Yaskawa INFORM job: malben_before.JBI

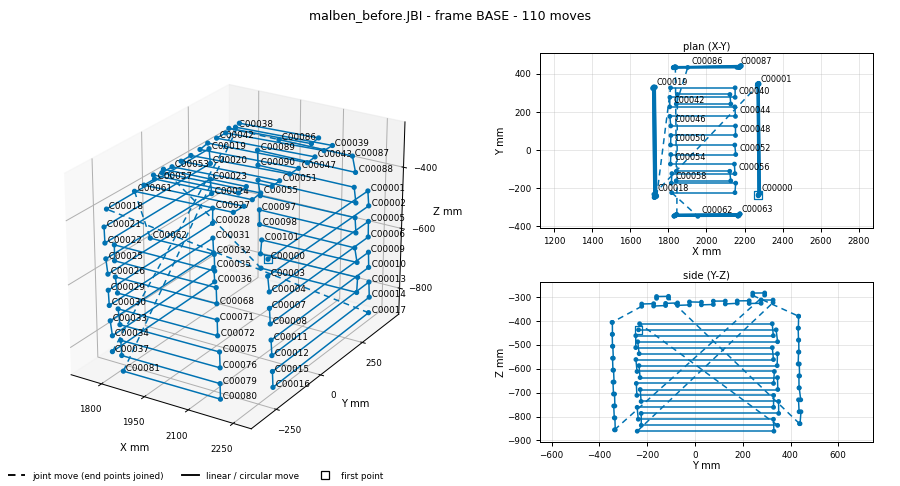
[picture p0: tool path of malben_before.JBI in frame BASE, 110 of 110 moves have a stored position in this frame; points joined in program order, loops and branches not executed]
/JOB
//NAME malben_before
//POS
///NPOS 110,0,0,0,0,0
///TOOL 0
///POSTYPE BASE
///RECTAN
///RCONF 1,0,0,0,0,0,0,0,0,0,0,0,0,0,0,0,0,0,0,0,0,0,0,0
C00000=2270.974700,-236.314400,-436.599200,0.000000,0.000000,0.000000
C00001=2266.659400,339.742100,-436.599200,0.000000,0.000000,0.000000
C00002=2267.434100,345.923800,-486.599200,0.000000,0.000000,0.000000
C00003=2272.441700,-239.676100,-486.599200,0.000000,0.000000,0.000000
C00004=2274.161000,-233.772700,-536.599200,0.000000,0.000000,0.000000
C00005=2268.116700,345.207300,-536.599200,0.000000,0.000000,0.000000
C00006=2269.414500,344.079000,-586.599200,0.000000,0.000000,0.000000
C00007=2275.422000,-234.403400,-586.599200,0.000000,0.000000,0.000000
C00008=2275.677100,-229.849900,-636.599200,0.000000,0.000000,0.000000
C00009=2270.908900,345.469500,-636.599200,0.000000,0.000000,0.000000
C00010=2272.247500,346.658600,-686.599200,0.000000,0.000000,0.000000
C00011=2278.345000,-229.368800,-686.599200,0.000000,0.000000,0.000000
C00012=2279.048100,-225.521500,-736.599200,0.000000,0.000000,0.000000
C00013=2272.572100,350.100400,-736.599200,0.000000,0.000000,0.000000
C00014=2274.809400,350.446800,-786.599200,0.000000,0.000000,0.000000
C00015=2281.061100,-225.219100,-786.599200,0.000000,0.000000,0.000000
C00016=2282.853200,-224.776000,-836.599200,0.000000,0.000000,0.000000
C00017=2276.307800,346.007400,-836.599200,0.000000,0.000000,0.000000
C00018=1724.578400,-231.807500,-411.083700,0.000000,90.000000,0.000000
C00019=1718.279300,323.447600,-411.083700,0.000000,90.000000,0.000000
C00020=1719.725400,327.955100,-461.083700,0.000000,90.000000,0.000000
C00021=1725.796900,-247.885600,-461.083700,0.000000,90.000000,0.000000
C00022=1727.476900,-248.031700,-511.083700,0.000000,90.000000,0.000000
C00023=1721.770500,323.709400,-511.083700,0.000000,90.000000,0.000000
C00024=1723.614500,328.610900,-561.083700,0.000000,90.000000,0.000000
C00025=1728.674900,-247.324100,-561.083700,0.000000,90.000000,0.000000
C00026=1731.265400,-242.598600,-611.083700,0.000000,90.000000,0.000000
C00027=1724.878400,332.404800,-611.083700,0.000000,90.000000,0.000000
C00028=1725.967100,328.907000,-661.083700,0.000000,90.000000,0.000000
C00029=1733.123300,-245.670000,-661.083700,0.000000,90.000000,0.000000
C00030=1733.584900,-243.188200,-711.083700,0.000000,90.000000,0.000000
C00031=1726.804300,329.270600,-711.083700,0.000000,90.000000,0.000000
C00032=1729.229800,328.994100,-761.083700,0.000000,90.000000,0.000000
C00033=1734.902000,-242.222300,-761.083700,0.000000,90.000000,0.000000
C00034=1737.913800,-237.463900,-811.083700,0.000000,90.000000,0.000000
C00035=1730.236300,328.580500,-811.083700,0.000000,90.000000,0.000000
C00036=1731.867100,330.516900,-861.083700,0.000000,90.000000,0.000000
C00037=1739.462300,-241.828500,-861.083700,0.000000,90.000000,0.000000
C00038=1812.070000,326.956500,-322.467000,-180.000000,0.000000,90.000000
C00039=2150.695600,326.956500,-312.028700,-180.000000,0.000000,90.000000
C00040=2150.727600,276.956500,-311.505300,-180.000000,0.000000,90.000000
C00041=1808.470300,276.956500,-325.644000,-180.000000,0.000000,90.000000
C00042=1807.754500,226.956500,-326.266200,-180.000000,0.000000,90.000000
C00043=2149.229600,226.956500,-314.851000,-180.000000,0.000000,90.000000
C00044=2152.427900,176.956500,-315.522800,-180.000000,0.000000,90.000000
C00045=1808.354700,176.956500,-325.499800,-180.000000,0.000000,90.000000
C00046=1813.127700,126.956500,-328.391500,-180.000000,0.000000,90.000000
C00047=2152.547100,126.956500,-316.102600,-180.000000,0.000000,90.000000
C00048=2152.688400,76.956500,-316.428000,-180.000000,0.000000,90.000000
C00049=1813.792200,76.956500,-330.537400,-180.000000,0.000000,90.000000
C00050=1812.079500,26.956500,-332.110200,-180.000000,0.000000,90.000000
C00051=2148.963600,26.956500,-320.940800,-180.000000,0.000000,90.000000
C00052=2153.965100,-23.043500,-319.751400,-180.000000,0.000000,90.000000
C00053=1813.274400,-23.043500,-332.397900,-180.000000,0.000000,90.000000
C00054=1811.443300,-73.043500,-334.201000,-180.000000,0.000000,90.000000
C00055=2146.917700,-73.043500,-323.945200,-180.000000,0.000000,90.000000
C00056=2149.738000,-123.043500,-326.004000,-180.000000,0.000000,90.000000
C00057=1819.062400,-123.043500,-334.939200,-180.000000,0.000000,90.000000
C00058=1816.212900,-173.043500,-337.150600,-180.000000,0.000000,90.000000
C00059=2153.683800,-173.043500,-327.184800,-180.000000,0.000000,90.000000
C00060=2149.816500,-223.043500,-328.439400,-180.000000,0.000000,90.000000
C00061=1817.967700,-223.043500,-338.250300,-180.000000,0.000000,90.000000
C00062=1954.986900,-347.317400,-405.440900,-90.000000,0.000000,0.000000
C00063=2165.301400,-346.003700,-405.440900,-90.000000,0.000000,0.000000
C00064=2166.306400,-345.533400,-455.440900,-90.000000,0.000000,0.000000
C00065=1831.008500,-346.423600,-455.440900,-90.000000,0.000000,0.000000
C00066=1829.824700,-345.452500,-505.440900,-90.000000,0.000000,0.000000
C00067=2169.877900,-343.987400,-505.440900,-90.000000,0.000000,0.000000
C00068=2170.261000,-341.942900,-555.440900,-90.000000,0.000000,0.000000
C00069=1830.845900,-345.180900,-555.440900,-90.000000,0.000000,0.000000
C00070=1835.840700,-343.537100,-605.440900,-90.000000,0.000000,0.000000
C00071=2170.679700,-340.902100,-605.440900,-90.000000,0.000000,0.000000
C00072=2170.579800,-338.805400,-655.440900,-90.000000,0.000000,0.000000
C00073=1836.308000,-343.283400,-655.440900,-90.000000,0.000000,0.000000
C00074=1839.916600,-341.222400,-705.440900,-90.000000,0.000000,0.000000
C00075=2175.279700,-336.688900,-705.440900,-90.000000,0.000000,0.000000
C00076=2176.238200,-335.487800,-755.440900,-90.000000,0.000000,0.000000
C00077=1840.835800,-340.227800,-755.440900,-90.000000,0.000000,0.000000
C00078=1841.292900,-337.885200,-805.440900,-90.000000,0.000000,0.000000
C00079=2175.716600,-335.286800,-805.440900,-90.000000,0.000000,0.000000
C00080=2175.900100,-333.842700,-855.440900,-90.000000,0.000000,0.000000
C00081=1845.052500,-336.997600,-855.440900,-90.000000,0.000000,0.000000
C00082=1847.834300,291.860000,-291.167300,-180.000000,0.000000,90.000000
C00083=2123.193800,291.860000,-282.202500,-180.000000,0.000000,90.000000
C00084=2127.968600,241.860000,-282.721100,-180.000000,0.000000,90.000000
C00085=1842.147700,241.860000,-292.609500,-180.000000,0.000000,90.000000
C00086=1902.222600,433.807700,-379.657800,90.000000,0.000000,0.000000
C00087=2160.048600,433.981200,-379.657800,90.000000,0.000000,0.000000
C00088=2172.433200,432.884400,-429.657800,90.000000,0.000000,0.000000
C00089=1826.230300,432.054000,-429.657800,90.000000,0.000000,0.000000
C00090=1827.301000,433.425300,-479.657800,90.000000,0.000000,0.000000
C00091=2168.117900,434.398200,-479.657800,90.000000,0.000000,0.000000
C00092=2174.981500,435.019500,-529.657800,90.000000,0.000000,0.000000
C00093=1827.672000,433.648700,-529.657800,90.000000,0.000000,0.000000
C00094=1837.169100,432.018700,-579.657800,90.000000,0.000000,0.000000
C00095=2172.360400,436.705800,-579.657800,90.000000,0.000000,0.000000
C00096=2175.918000,437.858200,-629.657800,90.000000,0.000000,0.000000
C00097=1832.142800,435.174100,-629.657800,90.000000,0.000000,0.000000
C00098=1832.804900,435.627000,-679.657800,90.000000,0.000000,0.000000
C00099=2173.854800,436.487800,-679.657800,90.000000,0.000000,0.000000
C00100=2179.550700,442.763800,-729.657800,90.000000,0.000000,0.000000
C00101=1842.051700,433.535700,-729.657800,90.000000,0.000000,0.000000
C00102=1836.410100,435.862900,-779.657800,90.000000,0.000000,0.000000
C00103=2182.210400,443.750100,-779.657800,90.000000,0.000000,0.000000
C00104=2182.276600,439.819200,-829.657800,90.000000,0.000000,0.000000
C00105=1837.285600,437.720700,-829.657800,90.000000,0.000000,0.000000
C00106=1842.355600,-110.852000,-303.697100,-180.000000,0.000000,90.000000
C00107=2122.511400,-110.852000,-296.331300,-180.000000,0.000000,90.000000
C00108=2127.898900,-160.852000,-297.180800,-180.000000,0.000000,90.000000
C00109=1841.572200,-160.852000,-304.679300,-180.000000,0.000000,90.000000
//INST
///DATE 2023/01/10 10:12
///ATTR SC,RW,RJ
////FRAME BASE
///GROUP1 RB1
NOP
MOVJ C00000 VJ=15.0
MOVL C00001 V=200.0
MOVL C00002 V=200.0
MOVL C00003 V=200.0
MOVL C00004 V=200.0
MOVL C00005 V=200.0
MOVL C00006 V=200.0
MOVL C00007 V=200.0
MOVL C00008 V=200.0
MOVL C00009 V=200.0
MOVL C00010 V=200.0
MOVL C00011 V=200.0
MOVL C00012 V=200.0
MOVL C00013 V=200.0
MOVL C00014 V=200.0
MOVL C00015 V=200.0
MOVL C00016 V=200.0
MOVL C00017 V=200.0
MOVJ C00018 VJ=15.0
MOVL C00019 V=200.0
MOVL C00020 V=200.0
MOVL C00021 V=200.0
MOVL C00022 V=200.0
MOVL C00023 V=200.0
MOVL C00024 V=200.0
MOVL C00025 V=200.0
MOVL C00026 V=200.0
MOVL C00027 V=200.0
MOVL C00028 V=200.0
MOVL C00029 V=200.0
MOVL C00030 V=200.0
MOVL C00031 V=200.0
MOVL C00032 V=200.0
MOVL C00033 V=200.0
MOVL C00034 V=200.0
MOVL C00035 V=200.0
MOVL C00036 V=200.0
MOVL C00037 V=200.0
MOVJ C00038 VJ=15.0
MOVL C00039 V=200.0
MOVL C00040 V=200.0
MOVL C00041 V=200.0
MOVL C00042 V=200.0
MOVL C00043 V=200.0
MOVL C00044 V=200.0
MOVL C00045 V=200.0
MOVL C00046 V=200.0
MOVL C00047 V=200.0
MOVL C00048 V=200.0
MOVL C00049 V=200.0
MOVL C00050 V=200.0
MOVL C00051 V=200.0
MOVL C00052 V=200.0
MOVL C00053 V=200.0
MOVL C00054 V=200.0
MOVL C00055 V=200.0
MOVL C00056 V=200.0
MOVL C00057 V=200.0
MOVL C00058 V=200.0
MOVL C00059 V=200.0
MOVL C00060 V=200.0
MOVL C00061 V=200.0
MOVJ C00062 VJ=15.0
MOVL C00063 V=200.0
MOVL C00064 V=200.0
MOVL C00065 V=200.0
MOVL C00066 V=200.0
MOVL C00067 V=200.0
MOVL C00068 V=200.0
MOVL C00069 V=200.0
MOVL C00070 V=200.0
MOVL C00071 V=200.0
MOVL C00072 V=200.0
MOVL C00073 V=200.0
MOVL C00074 V=200.0
MOVL C00075 V=200.0
MOVL C00076 V=200.0
MOVL C00077 V=200.0
MOVL C00078 V=200.0
MOVL C00079 V=200.0
MOVL C00080 V=200.0
MOVL C00081 V=200.0
MOVJ C00082 VJ=15.0
MOVL C00083 V=200.0
MOVL C00084 V=200.0
MOVL C00085 V=200.0
MOVJ C00086 VJ=15.0
MOVL C00087 V=200.0
MOVL C00088 V=200.0
MOVL C00089 V=200.0
MOVL C00090 V=200.0
MOVL C00091 V=200.0
MOVL C00092 V=200.0
MOVL C00093 V=200.0
MOVL C00094 V=200.0
MOVL C00095 V=200.0
MOVL C00096 V=200.0
MOVL C00097 V=200.0
MOVL C00098 V=200.0
MOVL C00099 V=200.0
MOVL C00100 V=200.0
MOVL C00101 V=200.0
MOVL C00102 V=200.0
MOVL C00103 V=200.0
MOVL C00104 V=200.0
MOVL C00105 V=200.0
MOVJ C00106 VJ=15.0
MOVL C00107 V=200.0
MOVL C00108 V=200.0
MOVL C00109 V=200.0
END
